{attribute 'linkalways'} 
{attribute 'no_explicit_call' := 'This FB is a CLASS and must be accessed using methods or properties'}
{attribute 'enable_dynamic_creation'}
FUNCTION_BLOCK JsonSerializer EXTENDS Disposable IMPLEMENTS I_Serializer;
VAR
	jsonSaxWriter : FB_JsonSaxWriter;
END_VAR

METHOD PUBLIC AddBase64 : I_Serializer
VAR_INPUT
	pBytes : POINTER TO BYTE;
	nBytes : DINT;
END_VAR
jsonSaxWriter.AddBase64(pBytes, nBytes);
AddBase64 := THIS^;
END_METHOD

METHOD PUBLIC AddBool : I_Serializer
VAR_INPUT
	Value : BOOL;
END_VAR
jsonSaxWriter.AddBool(Value);
AddBool := THIS^;
END_METHOD

METHOD PUBLIC AddByte : I_Serializer
VAR_INPUT
	Value : BYTE;
END_VAR
jsonSaxWriter.AddUDint(BYTE_TO_UDINT(Value));
AddByte := THIS^;
END_METHOD

METHOD PUBLIC AddBytesAsHex : I_Serializer
VAR_INPUT
	pBytes : POINTER TO BYTE;
	nBytes : DINT;
END_VAR
jsonSaxWriter.AddHexBinary(pBytes, nBytes);
AddBytesAsHex := THIS^;
END_METHOD

METHOD PUBLIC AddDateTime : I_Serializer
VAR_INPUT
	Value : DATE_AND_TIME;
END_VAR
jsonSaxWriter.AddDateTime(Value);
AddDateTime := THIS^;
END_METHOD

METHOD PUBLIC AddDcTime : I_Serializer
VAR_INPUT
	Value : DCTIME;
END_VAR
jsonSaxWriter.AddDcTime(Value);
AddDcTime := THIS^;
END_METHOD

METHOD PUBLIC AddDint : I_Serializer
VAR_INPUT
	Value : DINT;
END_VAR
jsonSaxWriter.AddDint(Value);
AddDint := THIS^;
END_METHOD

METHOD PUBLIC AddDword : I_Serializer
VAR_INPUT
	Value : DWORD;
END_VAR
jsonSaxWriter.AddUDint(DWORD_TO_UDINT(Value));
AddDword := THIS^;
END_METHOD

METHOD PUBLIC AddFileTime : I_Serializer
VAR_INPUT
	Value : FILETIME;
END_VAR
jsonSaxWriter.AddFileTime(Value);
AddFileTime := THIS^;
END_METHOD

METHOD PUBLIC AddInt : I_Serializer
VAR_INPUT
	Value : INT;
END_VAR
jsonSaxWriter.AddDint(INT_TO_DINT(Value));
AddInt := THIS^;
END_METHOD

METHOD PUBLIC AddKey : I_Serializer
VAR_INPUT
	Key : T_MAXSTRING;
END_VAR
jsonSaxWriter.AddKey(Key);
AddKey := THIS^;
END_METHOD

METHOD PUBLIC AddKeyBase64 : I_Serializer
VAR_INPUT
	Key : T_MAXSTRING;
	pBytes : POINTER TO BYTE;
	nBytes : DINT;
END_VAR
AddKey(Key);
AddBase64(pBytes, nBytes);
AddKeyBase64 := THIS^;
END_METHOD

METHOD PUBLIC AddKeyBool : I_Serializer
VAR_INPUT
	Key : T_MAXSTRING;
	Value : BOOL;
END_VAR
AddKey(Key);
AddBool(Value);
AddKeyBool := THIS^;
END_METHOD

METHOD PUBLIC AddKeyByte : I_Serializer
VAR_INPUT
	Key : T_MAXSTRING;
	Value : BYTE;
END_VAR
AddKey(Key);
AddByte(Value);
AddKeyByte := THIS^;
END_METHOD

METHOD PUBLIC AddKeyBytesAsHex : I_Serializer
VAR_INPUT
	Key : T_MAXSTRING;
	pBytes : POINTER TO BYTE;
	nBytes : DINT;
END_VAR
AddKey(Key);
AddBytesAsHex(pBytes, nBytes);
AddKeyBytesAsHex := THIS^;
END_METHOD

METHOD PUBLIC AddKeyDateTime : I_Serializer
VAR_INPUT
	Key : T_MAXSTRING;
	Value : DATE_AND_TIME;
END_VAR
AddKey(Key);
AddDateTime(Value);
AddKeyDateTime := THIS^;
END_METHOD

METHOD PUBLIC AddKeyDcTime : I_Serializer
VAR_INPUT
	Key : T_MAXSTRING;
	Value : DCTIME;
END_VAR
AddKey(Key);
AddDcTime(Value);
AddKeyDcTime := THIS^;
END_METHOD

METHOD PUBLIC AddKeyDint : I_Serializer
VAR_INPUT
	Key : T_MAXSTRING;
	Value : DINT;
END_VAR
AddKey(Key);
AddDint(Value);
AddKeyDint := THIS^;
END_METHOD

METHOD PUBLIC AddKeyDword : I_Serializer
VAR_INPUT
	Key : T_MAXSTRING;
	Value : DWORD;
END_VAR
AddKey(Key);
AddDword(Value);
AddKeyDword := THIS^;
END_METHOD

METHOD PUBLIC AddKeyFileTime : I_Serializer
VAR_INPUT
	Key : T_MAXSTRING;
	Value : FILETIME;
END_VAR
AddKey(Key);
AddFileTime(Value);
AddKeyFileTime := THIS^;
END_METHOD

METHOD PUBLIC AddKeyInt : I_Serializer
VAR_INPUT
	Key : T_MAXSTRING;
	Value : INT;
END_VAR
AddKey(Key);
AddInt(Value);
AddKeyInt := THIS^;
END_METHOD

METHOD PUBLIC AddKeyLint : I_Serializer
VAR_INPUT
	Key : T_MAXSTRING;
	Value : LINT;
END_VAR
AddKey(Key);
AddLint(Value);
AddKeyLint := THIS^;
END_METHOD

METHOD PUBLIC AddKeyLreal : I_Serializer
VAR_INPUT
	Key : T_MAXSTRING;
	Value : LREAL;
END_VAR
AddKey(Key);
AddLreal(Value);
AddKeyLreal := THIS^;
END_METHOD

METHOD PUBLIC AddKeyLtime : I_Serializer
VAR_INPUT
	Key : T_MAXSTRING;
	Value : LTIME;
END_VAR
AddKey(Key);
AddLTIME(Value);
AddKeyLtime := THIS^;
END_METHOD

METHOD PUBLIC AddKeyLword : I_Serializer
VAR_INPUT
	Key : T_MAXSTRING;
	Value : LWORD;
END_VAR
AddKey(Key);
AddLword(Value);
AddKeyLword := THIS^;
END_METHOD

METHOD PUBLIC AddKeyNull : I_Serializer
VAR_INPUT
	Key : T_MAXSTRING;
END_VAR
AddKey(Key);
AddNull();
AddKeyNull := THIS^;
END_METHOD

METHOD PUBLIC AddKeyRawObject : I_Serializer
VAR_INPUT
	Key : T_MAXSTRING;
	RawObject : REFERENCE TO STRING;;
END_VAR
AddKey(Key);
AddRawObject(RawObject);
AddKeyRawObject := THIS^;
END_METHOD

METHOD PUBLIC AddKeyReal : I_Serializer
VAR_INPUT
	Key : T_MAXSTRING;
	Value : REAL;
END_VAR
AddKey(Key);
AddReal(Value);
AddKeyReal := THIS^;
END_METHOD

METHOD PUBLIC AddKeySint : I_Serializer
VAR_INPUT
	Key : T_MAXSTRING;
	Value : SINT;
END_VAR
AddKey(Key);
AddSint(Value);
AddKeySint := THIS^;
END_METHOD

METHOD PUBLIC AddKeyString : I_Serializer
VAR_INPUT
	Key : T_MAXSTRING;
	Value : T_MAXSTRING;
END_VAR
AddKey(Key);
AddString(Value);
AddKeyString := THIS^;
END_METHOD

METHOD PUBLIC AddKeyStringByRef : I_Serializer
VAR_INPUT
	Key : T_MAXSTRING;
	Value : REFERENCE TO STRING;;
END_VAR
AddKey(Key);
AddStringByRef(Value);
AddKeyStringByRef := THIS^;
END_METHOD

METHOD PUBLIC AddKeyTime : I_Serializer
VAR_INPUT
	Key : T_MAXSTRING;
	Value : TIME;
END_VAR
AddKey(Key);
AddTime(Value);
AddKeyTime := THIS^;
END_METHOD

METHOD PUBLIC AddKeyTod : I_Serializer
VAR_INPUT
	Key : T_MAXSTRING;
	Value : TOD;
END_VAR
AddKey(Key);
AddTod(Value);
AddKeyTod := THIS^;
END_METHOD

METHOD PUBLIC AddKeyUdint : I_Serializer
VAR_INPUT
	Key : T_MAXSTRING;
	Value : UDINT;
END_VAR
AddKey(Key);
AddUdint(Value);
AddKeyUdint := THIS^;
END_METHOD

METHOD PUBLIC AddKeyUint : I_Serializer
VAR_INPUT
	Key : T_MAXSTRING;
	Value : UINT;
END_VAR
AddKey(Key);
AddUint(Value);
AddKeyUint := THIS^;
END_METHOD

METHOD PUBLIC AddKeyUlint : I_Serializer
VAR_INPUT
	Key : T_MAXSTRING;
	Value : ULINT;
END_VAR
AddKey(Key);
AddUlint(Value);
AddKeyUlint := THIS^;
END_METHOD

METHOD PUBLIC AddKeyUsint : I_Serializer
VAR_INPUT
	Key : T_MAXSTRING;
	Value : USINT;
END_VAR
AddKey(Key);
AddUsint(Value);
AddKeyUsint := THIS^;
END_METHOD

METHOD PUBLIC AddKeyWord : I_Serializer
VAR_INPUT
	Key : T_MAXSTRING;
	Value : WORD;
END_VAR
AddKey(Key);
AddWord(Value);
AddKeyWord := THIS^;
END_METHOD

METHOD PUBLIC AddLint : I_Serializer
VAR_INPUT
	Value : LINT;
END_VAR
jsonSaxWriter.AddLint(Value);
AddLint := THIS^;
END_METHOD

METHOD PUBLIC AddLreal : I_Serializer
VAR_INPUT
	Value : LREAL;
END_VAR
jsonSaxWriter.AddLreal(Value);
AddLreal := THIS^;
END_METHOD

METHOD PUBLIC AddLtime : I_Serializer
VAR_INPUT
	Value : LTIME;
END_VAR
VAR
	converted : T_MAXSTRING;
END_VAR
converted := LTIME_TO_STRING(Value);
jsonSaxWriter.AddString(converted);
AddLtime := THIS^;
END_METHOD

METHOD PUBLIC AddLword : I_Serializer
VAR_INPUT
	Value : LWORD;
END_VAR
jsonSaxWriter.AddUlint(LWORD_TO_ULINT(Value));
AddLword := THIS^;
END_METHOD

METHOD PUBLIC AddNull : I_Serializer
VAR_INPUT
END_VAR
jsonSaxWriter.AddNull();
AddNull := THIS^;
END_METHOD

METHOD PUBLIC AddRawObject
VAR_INPUT
	RawObject : REFERENCE TO STRING;
END_VAR
jsonSaxWriter.AddRawObject(RawObject);
END_METHOD

METHOD PUBLIC AddReal : I_Serializer
VAR_INPUT
	Value : REAL;
END_VAR
jsonSaxWriter.AddReal(Value);
AddReal := THIS^;
END_METHOD

METHOD PUBLIC AddSint : I_Serializer
VAR_INPUT
	Value : SINT;
END_VAR
jsonSaxWriter.AddDint(SINT_TO_DINT(Value));
AddSint := THIS^;
END_METHOD

METHOD PUBLIC AddString : I_Serializer
VAR_INPUT
	Value : T_MAXSTRING;
END_VAR
jsonSaxWriter.AddString(Value);
AddString := THIS^;
END_METHOD

METHOD PUBLIC AddStringByRef : I_Serializer
VAR_INPUT
	Value : REFERENCE TO STRING;
END_VAR
jsonSaxWriter.AddString(Value);
AddStringByRef := THIS^;
END_METHOD

METHOD PUBLIC AddTime : I_Serializer
VAR_INPUT
	Value : TIME;
END_VAR
VAR
	converted : T_MAXSTRING;
END_VAR
converted := TIME_TO_STRING(Value);
jsonSaxWriter.AddString(converted);
AddTime := THIS^;
END_METHOD

METHOD PUBLIC AddTod : I_Serializer
VAR_INPUT
	Value : TOD;
END_VAR
VAR
	converted : T_MAXSTRING;
END_VAR
converted := TOD_TO_STRING(Value);
jsonSaxWriter.AddString(converted);
AddTod := THIS^;
END_METHOD

METHOD PUBLIC AddUdint : I_Serializer
VAR_INPUT
	Value : UDINT;
END_VAR
jsonSaxWriter.AddUdint(Value);
AddUdint := THIS^;
END_METHOD

METHOD PUBLIC AddUint : I_Serializer
VAR_INPUT
	Value : UINT;
END_VAR
jsonSaxWriter.AddDint(UINT_TO_DINT(Value));
AddUint := THIS^;
END_METHOD

METHOD PUBLIC AddUlint : I_Serializer
VAR_INPUT
	Value : ULINT;
END_VAR
jsonSaxWriter.AddUlint(Value);
AddUlint := THIS^;
END_METHOD

METHOD PUBLIC AddUsint : I_Serializer
VAR_INPUT
	Value : USINT;
END_VAR
jsonSaxWriter.AddDint(USINT_TO_DINT(Value));
AddUsint := THIS^;
END_METHOD

METHOD PUBLIC AddWord : I_Serializer
VAR_INPUT
	Value : WORD;
END_VAR
jsonSaxWriter.AddUDint(WORD_TO_UDINT(Value));
AddWord := THIS^;
END_METHOD

METHOD PUBLIC Clone : I_Serializer
VAR
	pClone : POINTER TO JsonSerializer;
	jsonSize : UDINT;
	pJsonString : POINTER TO STRING;
END_VAR
pClone := __NEW(JsonSerializer);
Clone := pClone^;

jsonSize := jsonSaxWriter.GetDocumentLength();

IF jsonSize = 0 THEN
	// no further cloning to do. 
	RETURN;
END_IF

pJsonString := __NEW(BYTE, jsonSize);

IF jsonSaxWriter.CopyDocument(pJsonString^, jsonSize) = 0 THEN
	__DELETE(pJsonString);
	RETURN;
END_IF

pClone^.AddRawObject(pJsonString^);
__DELETE(pJsonString);
END_METHOD

METHOD PUBLIC EndArray : I_Serializer
VAR_INPUT
END_VAR
jsonSaxWriter.EndArray();
EndArray := THIS^;
END_METHOD

METHOD PUBLIC EndObject : I_Serializer
VAR_INPUT
END_VAR
jsonSaxWriter.EndObject();
EndObject := THIS^;
END_METHOD

METHOD FB_exit : BOOL
VAR_INPUT
	bInCopyCode : BOOL; // if TRUE, the exit method is called for exiting an instance that is copied afterwards (online change).
END_VAR
IF bInCopyCode THEN
	RETURN;
END_IF

jsonSaxWriter.ResetDocument();
END_METHOD

METHOD PUBLIC GetSeralizedDataLength : UDINT
VAR_INPUT
END_VAR
GetSeralizedDataLength := jsonSaxWriter.GetDocumentLength();
END_METHOD

METHOD PUBLIC Reset
VAR_INPUT
END_VAR
jsonSaxWriter.ResetDocument();
END_METHOD

METHOD PUBLIC StartArray : I_Serializer
VAR_INPUT
END_VAR
jsonSaxWriter.StartArray();
StartArray := THIS^;
END_METHOD

METHOD PUBLIC StartObject : I_Serializer
VAR_INPUT
END_VAR
jsonSaxWriter.StartObject();
StartObject := THIS^;
END_METHOD

METHOD TryCopySerialziedData : BOOL
VAR_INPUT
	DestinationAddress : PVOID;
	DestinationSize : UDINT;
END_VAR
VAR
	pString : POINTER TO STRING;
END_VAR
pString := DestinationAddress;
TryCopySerialziedData := jsonSaxWriter.CopyDocument(pString^, DestinationSize) > 0;
END_METHOD

METHOD TryGetSerialziedData : BOOL
VAR_INPUT
	DestinationAddress : PVOID;
	DestinationSize : UDINT;
END_VAR
VAR
	pString : POINTER TO STRING;
END_VAR
pString := DestinationAddress;

IF jsonSaxWriter.CopyDocument(pString^, DestinationSize) = 0 THEN
	RETURN;
END_IF

jsonSaxWriter.ResetDocument();
TryGetSerialziedData := TRUE;
END_METHOD

END_FUNCTION_BLOCK

(* stored: Version 1.1.0.1, ProductVersion 3.1.4024.12
   POU JsonSerializer: Id {a078a77d-919e-02c8-0175-c4fc65266934}, SpecialFunc None
   Folder Destructor: Id {3907011e-eb8f-0553-1e1c-e03005a7629b}
   Method AddBase64: Id {ad8af037-fae0-0c07-3c94-826b2377866d}
   Method AddBool: Id {6d90cde9-6354-0169-3fa9-5c145f652834}
   Method AddByte: Id {7ac92249-8951-48f6-b4ed-849570dc6883}
   Method AddBytesAsHex: Id {0600fb3e-8f5a-05f7-1e6d-d11206abcd70}
   Method AddDateTime: Id {8c7eda1b-5b14-0678-33ef-9b246b9f10f3}
   Method AddDcTime: Id {ca8ebe35-10b4-0223-0155-7f78d3fe519e}
   Method AddDint: Id {1d8f4b0a-bf9d-0848-2333-c22bd6bddcc8}
   Method AddDword: Id {2ae2202f-d1b1-40a6-9e2d-a8043670e211}
   Method AddFileTime: Id {86acc8ec-2231-086e-3898-e657f3706d24}
   Method AddInt: Id {5acf8d5e-3d1c-4b63-b4ac-44fdd3970622}
   Method AddKey: Id {c268998b-e7cd-00be-06cc-87de8a50e171}
   Method AddKeyBase64: Id {226dbd0b-8945-0b3c-2476-897d0ebe994e}
   Method AddKeyBool: Id {e615d07c-122f-0a0e-1133-4f5d49dab613}
   Method AddKeyByte: Id {818880e0-482a-42b5-8dd8-789871bdf896}
   Method AddKeyBytesAsHex: Id {173458d5-25d6-0464-0f08-29a6f4b6f67f}
   Method AddKeyDateTime: Id {599f79d7-dd42-012e-11d1-f6c38d6e3e4f}
   Method AddKeyDcTime: Id {1c72224f-0f0d-022b-39c7-d02401770d7e}
   Method AddKeyDint: Id {f763b7c8-1414-0717-0943-ea4e86763634}
   Method AddKeyDword: Id {540a79c2-cd71-4962-8cde-21b09e0bd9b9}
   Method AddKeyFileTime: Id {1e8cbdc0-9651-09ff-0ee6-4cf0d5198cf3}
   Method AddKeyInt: Id {c30684f4-f54b-40b0-aee7-8714bf71b484}
   Method AddKeyLint: Id {93a4b1b1-c548-0cc8-36a1-8bbc6f1f96e4}
   Method AddKeyLreal: Id {3de83c78-c0b8-07ba-0316-0e89d41fd0bb}
   Method AddKeyLtime: Id {43dcd259-0812-40bd-b3c6-0869a77f1a75}
   Method AddKeyLword: Id {f60b31a1-e59e-4fe0-b88b-8ab0c04de557}
   Method AddKeyNull: Id {320bb752-5a43-03fd-1b75-fc446c4d78a3}
   Method AddKeyRawObject: Id {f6f7ebe5-d7f8-4d7e-9b71-9fe9d524c1d2}
   Method AddKeyReal: Id {908060e9-3f04-0c29-3d32-837febc1c160}
   Method AddKeySint: Id {28e71021-149d-4d69-912a-a94f4979cd4e}
   Method AddKeyString: Id {cbb173c3-3393-4fa4-a216-452317a488d7}
   Method AddKeyStringByRef: Id {2a6eb483-f2b9-0b2e-3a13-83a40541e3d0}
   Method AddKeyTime: Id {18896a8a-1f0b-4012-8714-30a95ab09ad0}
   Method AddKeyTod: Id {276beeaa-d984-4b1c-a868-21b0f7c984ee}
   Method AddKeyUdint: Id {1fe7b2dd-f6c6-08a9-285c-5aebd0c2532a}
   Method AddKeyUint: Id {7d752c03-c810-4940-ad3a-6ae0a6895c2a}
   Method AddKeyUlint: Id {313d2467-c71e-0175-1248-a68a6acf4a68}
   Method AddKeyUsint: Id {96d5f31c-efd5-4c45-b997-98415597c7fe}
   Method AddKeyWord: Id {e0ac96a6-b75a-4b1a-8301-5484e49f2f9f}
   Method AddLint: Id {f6077592-9658-07e9-3ac1-5a9abfa6eb6a}
   Method AddLreal: Id {cb4b071a-b1a9-00fe-1eca-81f6114e0748}
   Method AddLtime: Id {81ce9111-d025-4f53-866b-38ebcbd87699}
   Method AddLword: Id {b05f59af-6688-43b3-bbde-4f7063d40394}
   Method AddNull: Id {25f68032-13b3-0c03-072e-c1eee07d407d}
   Method AddRawObject: Id {13b4569e-f550-016e-02ae-6e99a0c4d8af}
   Method AddReal: Id {d816e560-9bfd-09f2-2b2f-40fee09a3b9f}
   Method AddSint: Id {9135dcd0-b034-4920-b96b-65785a528cf5}
   Method AddString: Id {e17ac7cc-4de5-43d2-a31a-9b1e37f37211}
   Method AddStringByRef: Id {6f6487ff-8de1-0c91-2104-b6e952f67a16}
   Method AddTime: Id {eb9b17cd-508b-4789-b52e-d0719324deb7}
   Method AddTod: Id {821d8f4a-5930-42ad-9981-d88ff5fe30ff}
   Method AddUdint: Id {3ddc980b-9db8-0020-07a1-04f2bfb7aca7}
   Method AddUint: Id {10849fd8-6aac-441f-b541-b1fb5dfca322}
   Method AddUlint: Id {075fe558-9abc-0f4f-082e-4d7a6c6bd15e}
   Method AddUsint: Id {5302fd01-4f17-4a65-82f6-6b0210901378}
   Method AddWord: Id {c7113a83-eadb-4abf-9586-4b017d6e6527}
   Method Clone: Id {c51cbd07-1d68-0dcc-2a95-ab4b2cf0ac77}
   Method EndArray: Id {018bc96b-3949-05b8-20b4-f72fb4f7b925}
   Method EndObject: Id {9885dc13-2b73-0e77-102a-409239ef4a46}
   Method FB_exit: Id {3cb318ca-b325-0918-1741-6ba22e5f3ce1}
   Method GetSeralizedDataLength: Id {1c78c716-4a8c-0fc4-3c51-4fa2ff67c724}
   Method Reset: Id {c56165be-9bab-04d2-305e-f6b63f631e33}
   Method StartArray: Id {543e10ae-9cba-0f16-0502-2d80f68b1480}
   Method StartObject: Id {e62c9855-d4b2-0908-1c6b-0143452154bd}
   Method TryCopySerialziedData: Id {37c74c7b-1c2b-08a9-1aff-1f7d750f78ee}
   Method TryGetSerialziedData: Id {4c0f20e1-f625-0427-312a-8cd2e74bdfc6} *)
